Staubli VAL3: feedbackStatus.pgx

public program feedbackStatus(num x_nOutConnFlag)
begin

  // Do nothing
  // See start() program for more details

end
